// TIA Portal V17 export
// export: Created 2022-07-28T18:02:45.4996981Z, ExportSetting None, DisplayName Totally Integrated Automation Portal, DisplayVersion V17, DisplayName TIA Portal Openness, DisplayVersion V17, DisplayName TIA Portal Teamcenter Gateway, DisplayVersion V17, DisplayName TIA Portal Version Control Interface, DisplayVersion V17, DisplayName TIA Portal Test Suite Advanced, DisplayVersion V17, DisplayName SINAMICS Startdrive Advanced, DisplayVersion V17, DisplayName SINAMICS DCC, DisplayVersion V17, DisplayName SINAMICS Startdrive G130, G150, S120, S150, SINAMICS MV, S210, DisplayVersion V17, DisplayName SINAMICS Startdrive G110M, G120, G120C, G120D, G120P, G115D, DisplayVersion V17, DisplayName STEP 7 Professional, DisplayVersion V17, DisplayName SIMATIC Energy Suite, DisplayVersion V17, DisplayName STEP 7 CFC, DisplayVersion V17, DisplayName STEP 7 Safety, DisplayVersion V17, DisplayName WinCC Advanced / Unified PC, DisplayVersion V17, DisplayName SIMATIC Visualization Architect, DisplayVersion V17
FUNCTION "Lib_FC_GenMoto_SwitchMode" : Void   // FC12, SCL
{ S7_Optimized_Access := 'TRUE' }
// stored: SetENOAutomatically false
   VAR_INPUT
      I_ManLocalModeActive : Bool;   // Switching in external mode ManualLocal if PRM.ManLocalPirority=1(hight)
   END_VAR
   VAR_IN_OUT
      IQI_CMD_Logic : Int;   // Command for use in logic
      IQ_Mode : "UDT_Mode";   // Current mode
      IQ_ObjDataConfig : Variant;   // Object data for use in program
      IQ_BUpDataConfig : Variant;   // Backup data for store simulation
      IQ_ObjDataCounters : Variant;   // Object data for use in program
      IQ_BUpDataCounters : Variant;   // Backup data for store simulation
   END_VAR
   VAR_TEMP
      t_InternalData : "Lib_UDT_Int";
      t_Buffer : Array[0..100] of Byte;
   END_VAR
BEGIN
   //Set internal data
   REGION Internal data
       #t_InternalData.AlwTrue := true;
       #t_InternalData.AlwFalse := false;
       #t_InternalData.i_Alw0 := 0;
       #t_InternalData.b_Alw0 := b#16#0;
       #t_InternalData.w_Alw0 := w#16#0;
       #t_InternalData.d_Alw0 := dw#16#0;
   END_REGION

   //Control simulation mode
   CASE #IQI_CMD_Logic OF
       7:  //Switch on simulation mode
           IF NOT #IQ_Mode.Simulation
           THEN
               #IQ_Mode.Simulation := true;

               //BackUp object data
               #t_InternalData.di_Tmp := 0;
               #t_InternalData.i_Tmp := Serialize(SRC_VARIABLE := #IQ_ObjDataConfig, DEST_ARRAY => #t_Buffer, POS := #t_InternalData.di_Tmp);

               #t_InternalData.di_Tmp := 0;
               #t_InternalData.i_Tmp := Deserialize(SRC_ARRAY := #t_Buffer, DEST_VARIABLE => #IQ_BUpDataConfig, POS := #t_InternalData.di_Tmp);

               #t_InternalData.di_Tmp := 0;
               #t_InternalData.i_Tmp := Serialize(SRC_VARIABLE := #IQ_ObjDataCounters, DEST_ARRAY => #t_Buffer, POS := #t_InternalData.di_Tmp);

               #t_InternalData.di_Tmp := 0;
               #t_InternalData.i_Tmp := Deserialize(SRC_ARRAY := #t_Buffer, DEST_VARIABLE => #IQ_BUpDataCounters, POS := #t_InternalData.di_Tmp); 

           END_IF;

       8:  //Switch off simulation mode
           IF #IQ_Mode.Simulation
           THEN
               #IQ_Mode.Simulation := FALSE;

               //Store object data from simulation backup
               #t_InternalData.di_Tmp := 0;
               #t_InternalData.i_Tmp := Serialize(SRC_VARIABLE := #IQ_BUpDataConfig, DEST_ARRAY => #t_Buffer, POS := #t_InternalData.di_Tmp);

               #t_InternalData.di_Tmp := 0;
               #t_InternalData.i_Tmp := Deserialize(SRC_ARRAY := #t_Buffer, DEST_VARIABLE => #IQ_ObjDataConfig, POS := #t_InternalData.di_Tmp);

               #t_InternalData.di_Tmp := 0;
               #t_InternalData.i_Tmp := Serialize(SRC_VARIABLE := #IQ_BUpDataCounters, DEST_ARRAY => #t_Buffer, POS := #t_InternalData.di_Tmp);

               #t_InternalData.di_Tmp := 0;
               #t_InternalData.i_Tmp := Deserialize(SRC_ARRAY := #t_Buffer, DEST_VARIABLE => #IQ_ObjDataCounters, POS := #t_InternalData.di_Tmp);

               #IQI_CMD_Logic := 31;
           END_IF;
       ELSE
           ;
   END_CASE;

   //Control technologie modes
   IF NOT #IQ_Mode.Repair
   THEN
       CASE #IQI_CMD_Logic OF

           1:  //Switch to manual remote mode
               #IQ_Mode.Disable := false;
               #IQ_Mode.Auto := false;
               #IQ_Mode.ManualLocal := false;
               #IQ_Mode.Service := false;
               #IQ_Mode.ManualRemote := true;

           2:  //Switch to auto mode
               #IQ_Mode.Disable := false;
               #IQ_Mode.ManualRemote := false;
               #IQ_Mode.ManualLocal := false;
               #IQ_Mode.Service := false;
               #IQ_Mode.Auto := true;

           3:  //Switch to manual local mode
               #IQ_Mode.Disable := false;
               #IQ_Mode.ManualRemote := false;
               #IQ_Mode.Auto := false;
               #IQ_Mode.Service := false;
               #IQ_Mode.ManualLocal := true;

           4:  //Switch to service mode
               #IQ_Mode.Disable := false;
               #IQ_Mode.Auto := false;
               #IQ_Mode.ManualLocal := false;
               #IQ_Mode.ManualRemote := true;
               #IQ_Mode.Service := true;

           5:  //Switch to repair mode (outputs disabled)
               #IQ_Mode.Disable := TRUE;
               #IQ_Mode.ManualRemote := false;
               #IQ_Mode.Auto := false;
               #IQ_Mode.Service := false;
               #IQ_Mode.ManualLocal := false;
               #IQ_Mode.Repair := true;

           10:  //Switch to disable mode (outputs disabled)
               #IQ_Mode.ManualRemote := false;
               #IQ_Mode.Auto := false;
               #IQ_Mode.Service := false;
               #IQ_Mode.ManualLocal := false;
               #IQ_Mode.Disable := true;
           ELSE
               ;
       END_CASE;
   ELSE
       CASE #IQI_CMD_Logic OF
           6:  //Switch off repair mode
               #IQ_Mode.Disable := true;
               #IQ_Mode.Repair := false;
           ELSE
               ;
       END_CASE;
   END_IF;

   //Switch to manual local mode from input
   IF #I_ManLocalModeActive
   THEN
       #IQ_Mode.Disable := false;
       #IQ_Mode.ManualRemote := false;
       #IQ_Mode.Auto := false;
       #IQ_Mode.Service := false;
       #IQ_Mode.ManualLocal := true;
   END_IF;

   //Switchon disable mode when not active other
   IF NOT #IQ_Mode.Disable
       AND NOT #IQ_Mode.ManualRemote
       AND NOT #IQ_Mode.Auto
       AND NOT #IQ_Mode.ManualLocal
       AND NOT #IQ_Mode.Service
       AND NOT #IQ_Mode.Repair
   THEN
       #IQ_Mode.Disable := true;
   END_IF;
END_FUNCTION
